(* CoDeSys 2.3.9.50 project: Sample01.pro *)
(* Libraries: STANDARD.LIB 5.6.98 11:03:02 *)

(* Task configuration *)
TASK Standard (PRIORITY := 0, INTERVAL := T#10ms);
	MAIN
END_TASK

(* POU MAIN, ST *)
PROGRAM MAIN
VAR
 PLCVar : ARRAY [0..99] OF INT;
  Index: BYTE;
 Total: BYTE;

END_VAR
FOR Index := 0 TO Total DO
  PLCVar[Index] := 3500 + INDEX  + Total;
END_FOR
END_PROGRAM

(* POU Ladder, LD *)
PROGRAM Ladder
VAR
	In1 AT %IX0.0:BOOL;

	Out1 AT %QX0.0: BOOL;
END_VAR
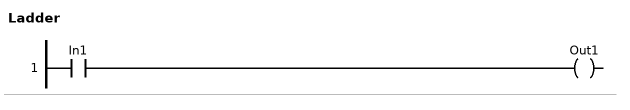
_LD_ (* Ladder Diagram *)
NETWORK 1
	[In1] --- (Out1)
_END_LD_
(* the same logic as Structured Text *)
(* Network 1 *)
Out1 := In1;
END_PROGRAM
